PROGRAM p_MPSSup
VAR
	q_xMFX_LENS_MPSOK: BOOL;
	BEAT: Heartbeat;

END_VAR

//Instantiate Heartbeat and check to see if IOC is alive
BEAT(BEAT:=i_xIOC_HEARTBEAT,DEADTIME:=TIME#1.0S);
q_xHEARTBEAT_ALIVE := BEAT.ALIVE;
IF NOT BEAT.ALIVE THEN
	q_xMFX_LENS_MPSOK := 0;
	q_xFAULTED := 0;
	RETURN;
END_IF

//Check no lens is unknown position
q_xLENSES_KNOWN := (   i_xMFX_LENS02.KNOWN   //i_xMFX_LENS01.KNOWN AND i_xMFX_LENS02.KNOWN
				 	   AND i_xMFX_LENS03.KNOWN 
				       AND i_xMFX_LENS04.KNOWN AND i_xMFX_LENS05.KNOWN 
					   AND i_xMFX_LENS06.KNOWN AND i_xMFX_LENS07.KNOWN
					   AND i_xMFX_LENS08.KNOWN AND i_xMFX_LENS09.KNOWN
					   AND i_xMFX_LENS10.KNOWN AND i_xXRT_LENS01.KNOWN
					   AND i_xXRT_LENS02.KNOWN AND i_xXRT_LENS03.KNOWN);
				
IF NOT q_xLENSES_KNOWN THEN
  q_xMFX_LENS_MPSOK := 0;
  q_xFAULTED := 1;
  RETURN;
END_IF

//Determine which lens group/s are being used
q_xMFX_LENSES_IN :=  i_xMFX_LENS02.IN  //i_xMFX_LENS01.IN OR i_xMFX_LENS02.IN
				 	 OR i_xMFX_LENS03.IN OR i_xMFX_LENS04.IN 
					 OR i_xMFX_LENS05.IN OR i_xMFX_LENS06.IN
					 OR i_xMFX_LENS07.IN OR i_xMFX_LENS08.IN
					 OR i_xMFX_LENS09.IN OR i_xMFX_LENS10.IN;

q_xXRT_LENSES_IN :=  i_xXRT_LENS01.IN 
				     OR i_xXRT_LENS02.IN
					 OR i_xXRT_LENS03.IN;


//If Both lenses are used, compare to pre-focused limit
IF q_xMFX_LENSES_IN AND q_xXRT_LENSES_IN THEN
	q_iLIMIT_MODE := 3;
	IF  i_rPREFOCUS_LIMIT > i_rBEAM_FOCUS THEN
		q_xMFX_LENS_MPSOK := 1;
		q_xFAULTED := 0;
	ELSE
		q_xMFX_LENS_MPSOK := 0;
		q_xFAULTED := 1;
	END_IF

//If only MFX lenses are in compare to MFX only limit
ELSIF q_xMFX_LENSES_IN THEN
	q_iLIMIT_MODE := 2;
	IF i_rMFX_ONLY_LIMIT > i_rBEAM_FOCUS THEN
		q_xMFX_LENS_MPSOK := 1;
		q_xFAULTED := 0;
	ELSE
		q_xMFX_LENS_MPSOK := 0;
		q_xFAULTED := 1;
	END_IF

//If only XRT lenses are in compare to XRT only limit
ELSIF q_xXRT_LENSES_IN THEN
	q_iLIMIT_MODE := 1;
	q_rCURRENT_LIMIT := i_rXRT_ONLY_LIMIT;
	IF i_rXRT_ONLY_LIMIT < i_rBEAM_FOCUS THEN
		q_xMFX_LENS_MPSOK := 1;
		q_xFAULTED := 0;
	ELSE
		q_xMFX_LENS_MPSOK := 0;
		q_xFAULTED := 1;
	END_IF
//IF no lenses are in, simply return 
ELSE 
	q_iLIMIT_MODE :=0;
	q_rCURRENT_LIMIT := 0.0;
	q_xMFX_LENS_MPSOK := 1;
	q_xFAULTED := 0;
	RETURN;
END_IF

END_PROGRAM

(* stored: Version 1.1.0.1, ProductVersion 3.1.4018.5
   POU p_MPSSup: Id {22fa257d-fc87-4b8c-8293-563a03fa02d7}, SpecialFunc None *)
